// TwinCAT 3 PLC project main
// ProgramVersion: 3.1.4024.0
// libraries:
//   Tc2_Standard, * (Beckhoff Automation GmbH)
//   Tc2_System, * (Beckhoff Automation GmbH)
//   Tc3_Module, * (Beckhoff Automation GmbH)
// project tree:
//   / GlobalTextList.TcGTLO, PlcTask.TcTTO, Visualization Manager.TcVMO (not stored)
//   POUs/ MAIN.TcPOU
//   VISUs/ Visu.TcVIS
// real-time tasks:
//   TASK PlcTask: cycle T#10ms, priority 20, ADS port 350

CONFIGURATION main
    RESOURCE PLC ON TwinCAT3
        TASK PlcTask(INTERVAL := T#10ms, PRIORITY := 20);
        PROGRAM MAIN WITH PlcTask : MAIN;
    END_RESOURCE
END_CONFIGURATION

// ---- POUs/MAIN.TcPOU
PROGRAM MAIN
VAR
	Q01 : BOOL;
	S01 : BOOL;
END_VAR

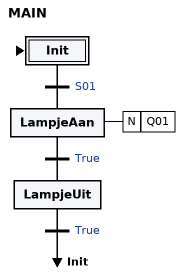
INITIAL_STEP Init:
END_STEP
TRANSITION FROM Init TO LampjeAan
    := S01;
END_TRANSITION
STEP LampjeAan:  // min time t#700ms
    Q01(N);
END_STEP
TRANSITION FROM LampjeAan TO LampjeUit
    := True;
END_TRANSITION
STEP LampjeUit:  // min time t#300ms
END_STEP
TRANSITION FROM LampjeUit TO Init
    := True;
END_TRANSITION

END_PROGRAM

// ---- VISUs/Visu.TcVIS
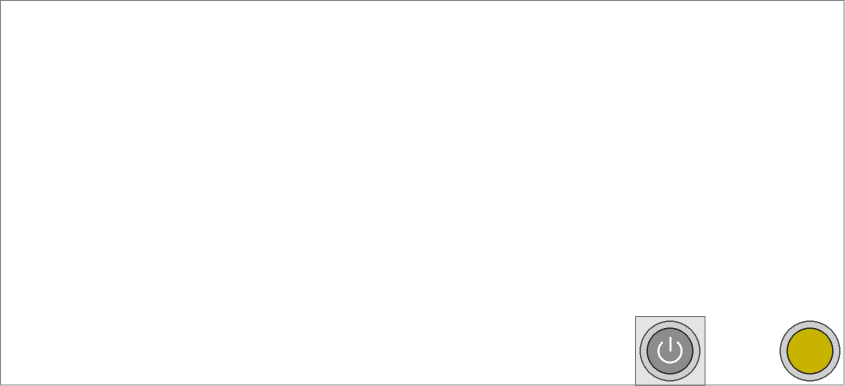
VISUALIZATION Visu  // 845x386
    Lamp1 (775,316 70x70), variable: MAIN.Q01, style: Lamp-Lamp1-Yellow
    PowerSwitch (635,316 70x70), variable: MAIN.S01, behaviour: TOGGLE, style: Switch-PowerSwitch-Gray
END_VISUALIZATION
